PROGRAM MAIN
VAR
END_VAR

END_PROGRAM

(* stored: Version 1.1.0.1, ProductVersion 3.1.0.12
   POU MAIN: Id {1b849b8a-729e-4d34-8fad-6f20c321f37d} *)
